RESOURCE_TYPE top
  (* Standard: 61499-2 *)
  (* Version 0.1, 2017-00-25, hpea485, UOA *)
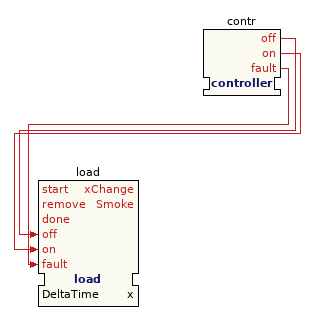
  FBS
    load : load;
    contr : controller;
  END_FBS
  EVENT_CONNECTIONS
    contr.off TO load.off;
    contr.on TO load.on;
    contr.fault TO load.fault;
  END_CONNECTIONS
END_RESOURCE_TYPE
